Staubli VAL3: recursion.pgx

program recursion()
  local string l_sItem
begin
  nNum=nNum+1
  delay(0.1)
  call recursion()

end
